RoboDK station: 3D_Orientation.rdk

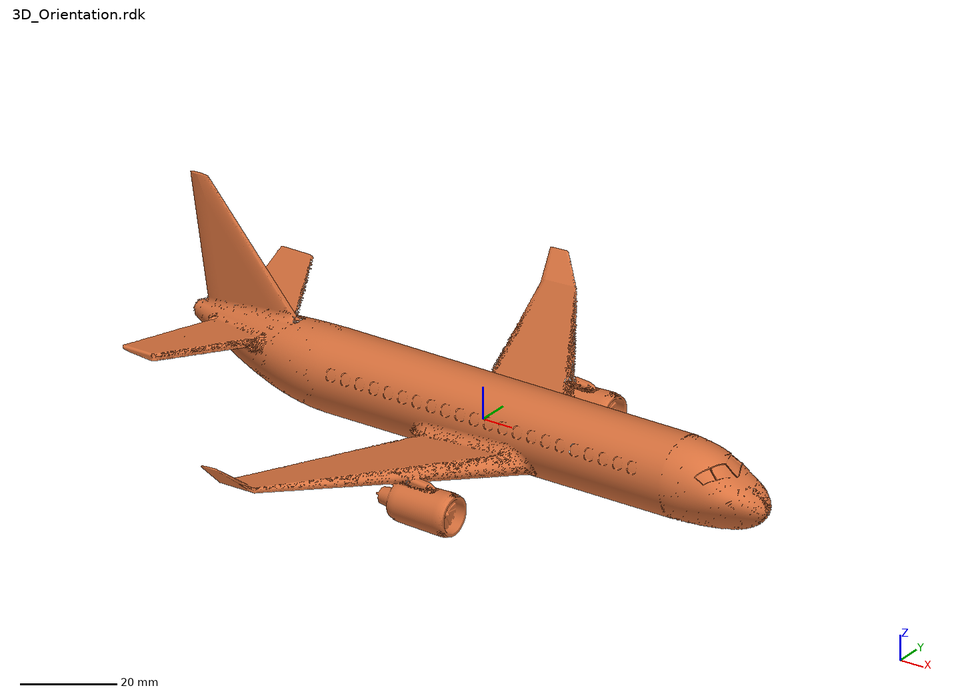
[picture v0: the station drawn from its stored meshes, robots at their saved joint values, targets as dots, program paths as lines]
Station 3D_Orientation (saved by RoboDK 5.7.4). Poses are relative to the parent item; angles as X-Y-Z fixed-axis rotations.
  - object plane at (0, 0, 0) mm, size 145.5 x 126 x 48.3 mm, geometry from plane.stl
  - object surgical_needle at (0, 0, 0) mm, size 36.5 x 50.2 x 4.5 mm, geometry from surgical_needle1.stl
  - frame world at (0, 0, 0) mm
